TYPE ST_LogBuffer :
STRUCT
    aEntries : ARRAY[1..100] OF ST_LogEntry;
END_STRUCT
END_TYPE

(* stored: Version 1.1.0.1
   DUT ST_LogBuffer: Id {93eb5be0-7697-48e2-8222-3bc985371d80} *)
